Fanuc KAREL source: kt00869.KL

-- PROVISIONAL review KL for V1013-1; original PC SHA256 ef4f89d89e6884a45988e103004d544c43e37e60b8a394771e0d4d690824865f
-- Incomplete behavior may be omitted. Consult companion uncertainty JSON. Do not deploy.
PROGRAM KT00869
%NOLOCKGROUP
VAR
  I1 : INTEGER
  I2 : INTEGER
  OUT : REAL
BEGIN
  -- UNRESOLVED_PC offsets 5-16; opcodes 2E,23
  -- UNRESOLVED_PC offsets 21-32; opcodes 2E,23
  -- UNRESOLVED_PC offsets 37-48; opcodes 2E,23
  -- UNRESOLVED_PC offsets 53-64; opcodes 2E,23
  -- UNRESOLVED_PC offsets 69-87; opcodes 27,27,21,64,76,64,23
  -- UNRESOLVED_PC offsets 92-96; opcodes 7F
END KT00869
